{attribute 'hide_all_locals'}
FUNCTION_BLOCK FB_RxMapper //See ST_RxMapping for more info.
VAR_INPUT
	bRun					: BOOL;
	bAutoCreateMappings		: BOOL; //Be careful with this, can quickly cause the Rx Mapper to use a lot of CPU time. This can lead to cycle exceeds. Configure CAN Interface RxFilter is recommeded if used!
	pCanItfHelper 			: POINTER TO FB_CanItfHelper;
	cbCanItfHelperSize		: UDINT; 
	paMappingData 			: POINTER TO ARRAY[0..65535] OF ST_RxMapping;
	cbMappingDataSize		: UDINT;
END_VAR
VAR_OUTPUT
	bBusy 					: BOOL;
	bError					: BOOL;
	eRxMapperHResult 		: E_CanRxMapperHResult;
	nMappingCnt				: UDINT;
END_VAR
VAR
	bUnmappedCanMsg			: BOOL;
	nRxMapperUpperIndex		: UDINT;
	nCobidtemp				: UDINT;
	nPrevRxCounter 			: UINT;
	index 					: UINT;
	stTempCanMsg			: ST_CanMsg;
	nMappingIndex 			: UDINT;
	CanHelperHResult		: E_CanItfHelperHResult;
END_VAR

IF NOT bRun THEN
	bBusy := FALSE;
	RETURN;
ELSE
	bBusy := TRUE;
END_IF

eRxMapperHResult := mCheckSetup();
IF (eRxMapperHResult < 0 ) THEN
	bError := TRUE;
	RETURN;
END_IF

eRxMapperHResult := E_CanRxMapperHResult.NoError;

nRxMapperUpperIndex := (cbMappingDataSize / SIZEOF(ST_RxMapping))-1;

FOR index:=0 TO GVL_CanItfHelper.nRxQueueUpperIndex BY 1 DO
	MEMSET(destAddr := ADR(stTempCanMsg), 0, n:=SIZEOF(stTempCanMsg));
	CanHelperHResult := pCanItfHelper^.mRxMessageGet(bGetRemove := TRUE, pRxCanMessage := ADR(stTempCanMsg));
	IF CanHelperHResult >= 0 THEN
		bUnmappedCanMsg := TRUE; //used later
		FOR nMappingIndex:= 0 TO MIN(nMappingCnt-1 , nRxMapperUpperIndex) BY 1 DO
			IF (paMappingData^[nMappingIndex].i_stCanMsg.CanHeader.nCobid = stTempCanMsg.CanHeader.nCobid) AND (paMappingData^[nMappingIndex].i_stCanMsg.CanHeader.bExtendedAddress = stTempCanMsg.CanHeader.bExtendedAddress) AND (paMappingData^[nMappingIndex].i_stCanMsg.CanHeader.bRTR = stTempCanMsg.CanHeader.bRTR) THEN
				bUnmappedCanMsg := FALSE;
				IF paMappingData^[nMappingIndex].i_bRun THEN
					IF 	(paMappingData^[nMappingIndex].i_pDestAddr <> 0) AND 
						(paMappingData^[nMappingIndex].i_cbDestSize <> 0) AND 
						(paMappingData^[nMappingIndex].i_cbDestSize >= UINT_TO_UDINT(stTempCanMsg.CanHeader.nMsgLength)) THEN
							paMappingData^[nMappingIndex].i_stCanMsg := stTempCanMsg;
							MEMCPY(paMappingData^[nMappingIndex].i_pDestAddr ,ADR(paMappingData^[nMappingIndex].i_stCanMsg.CanData[0]), paMappingData^[nMappingIndex].i_stCanMsg.CanHeader.nMsgLength);
							paMappingData^[nMappingIndex].o_bBusy := TRUE;
							paMappingData^[nMappingIndex].o_nUpdateCount := paMappingData^[nMappingIndex].o_nUpdateCount +1;					
					ELSE
						paMappingData^[nMappingIndex].o_bError := TRUE;
						eRxMapperHResult := E_CanRxMapperHResult.RxMappingHasError;
					END_IF					
				END_IF
			END_IF
		END_FOR
		IF bUnmappedCanMsg AND bAutoCreateMappings THEN
			eRxMapperHResult := THIS^.mCreateMsgMapping(bRun:=FALSE, stCanMsg:= stTempCanMsg,pDestAddr:= 0, cbDestSize := 0);
		END_IF
	END_IF
END_FOR

METHOD mAddMapping : E_CanRxMapperHResult
VAR_INPUT
	stInput		: ST_RxMapping;
END_VAR
mAddMapping := mCheckSetup();
IF (mAddMapping < 0 ) THEN
	bError := TRUE;
	RETURN;
END_IF

nRxMapperUpperIndex := (cbMappingDataSize / SIZEOF(ST_RxMapping))-1;

IF ((nMappingCnt > nRxMapperUpperIndex) OR (cbMappingDataSize = 0)) THEN
	mAddMapping := E_CanRxMapperHResult.RxMappingsListFull;
	RETURN;
END_IF

IF (stInput.i_bRun = FALSE) THEN
	mAddMapping := E_CanRxMapperHResult.RxMappingNotRunning;
END_IF

IF stInput.i_cbDestSize < stInput.i_stCanMsg.CanHeader.nMsgLength THEN
	mAddMapping := E_CanRxMapperHResult.RxMappingDestSizeError;
END_IF

IF (stInput.i_pDestAddr = 0) THEN
	mAddMapping := E_CanRxMapperHResult.RxMappingDestPointerError;
END_IF

paMappingData^[nMappingCnt] := stInput;
nMappingCnt := nMappingCnt + 1;
END_METHOD

METHOD PRIVATE mCheckSetup : E_CanRxMapperHResult
VAR_INPUT
END_VAR
IF ((cbMappingDataSize = 0) OR (paMappingData = 0)) THEN
	mCheckSetup := E_CanRxMapperHResult.MappingSetupIsInvalid;
	RETURN;
END_IF

IF ((pCanItfHelper = 0) OR (cbCanItfHelperSize <> SIZEOF(FB_CanItfHelper)))  THEN
	bError := TRUE;
	mCheckSetup := E_CanRxMapperHResult.RxMapperHasInvalidSetup;
	RETURN;
END_IF

IF (NOT pCanItfHelper^.bValidSetup) THEN
	mCheckSetup := E_CanRxMapperHResult.RxMapperHasInvalidSetup;
	RETURN;
END_IF
END_METHOD

METHOD mClearMappings : E_CanRxMapperHResult // clears all mappings paMappingData points to. Result always 0 NoError
VAR_INPUT
END_VAR
mClearMappings := mCheckSetup();
IF (mClearMappings < 0 ) THEN
	bError := TRUE;
	RETURN;
END_IF


mClearMappings := E_CanRxMapperHResult.NoError;
MEMSET(destAddr := ADR(paMappingData^), 0 , n:= SIZEOF(cbMappingDataSize)); //Pointer is to an array varaible, which is also a pointer. Clear the array not the array pointer.
nMappingCnt := 0;
END_METHOD

METHOD mCreateMsgMapping : E_CanRxMapperHResult
VAR_INPUT
	bRun: BOOL;
	stCanMsg : ST_CanMsg;
	pDestAddr : POINTER TO BYTE;
	cbDestSize	: UDINT;
END_VAR
VAR
	temp: ST_RxMapping;
END_VAR
mCreateMsgMapping := E_CanRxMapperHResult.NoError;

temp.i_bRun := bRun;
temp.i_stCanMsg := stCanMsg;
temp.i_pDestAddr := pDestAddr;
temp.i_cbDestSize:= cbDestSize;

mCreateMsgMapping := This^.mAddMapping(temp);
END_METHOD

METHOD mCreateNewMapping : E_CanRxMapperHResult
VAR_INPUT
	bRun: BOOL;
	nCobid : DWORD;
	nMsgLength : UINT;
	pDestAddr : POINTER TO BYTE;
	cbDestSize	: UDINT;
END_VAR
VAR
	temp: ST_RxMapping;
END_VAR
mCreateNewMapping := E_CanRxMapperHResult.NoError;

temp.i_bRun := bRun;
temp.i_stCanMsg.CanHeader.nCobid := nCobid;
temp.i_stCanMsg.CanHeader.nMsgLength := nMsgLength;
temp.i_pDestAddr := pDestAddr;
temp.i_cbDestSize:= cbDestSize;

mCreateNewMapping := This^.mAddMapping(temp);
END_METHOD

METHOD mSetMappingCnt : E_CanRxMapperHResult  // return true if successful, must be less then or equal to size of mapping array.
VAR_INPUT
	input : UDINT;
END_VAR
mSetMappingCnt := mCheckSetup();
IF (mSetMappingCnt < 0 ) THEN
	bError := TRUE;
	RETURN;
END_IF

nRxMapperUpperIndex := (cbMappingDataSize / SIZEOF(ST_RxMapping))-1;

IF input > nRxMapperUpperIndex THEN
	nMappingCnt := input;
	mSetMappingCnt := E_CanRxMapperHResult.InvalidParameter;
END_IF
END_METHOD

END_FUNCTION_BLOCK

(* stored: Version 1.1.0.1, ProductVersion 3.1.4024.11
   POU FB_RxMapper: Id {ea900807-319e-44b8-ac4e-e45598fef5bb}, SpecialFunc None
   Method mAddMapping: Id {9ed2d0bb-c61a-45d3-9723-0170ef273496}
   Method mCheckSetup: Id {9d53f300-9290-47b9-925c-e825ea4211d3}
   Method mClearMappings: Id {5b5ed598-1cdc-4fb8-b23d-db46c556d4e1}
   Method mCreateMsgMapping: Id {aac49f03-2daf-4432-a68c-4e36c2f43d05}
   Method mCreateNewMapping: Id {b9ef7bd9-0c1b-422b-8f62-a64cdae4fb4f}
   Method mSetMappingCnt: Id {1c9d09e7-bb4b-4a1b-befc-693c7d7043df} *)
